// TIA Portal V20 export
TYPE "typeStationDataReelCutInspection"
   STRUCT
      "Intro cut count 1" : DInt;   // Cnt
      "Introcut Vision - Tab length 1" : Real;   // mm
      "Introcut Vision - Tab height 1" : Real;   // mm
      "Introcut Vision - Electrode length 1" : Real;   // mm
      "Introcut Vision - Electrode height 1" : Real;   // mm
      "Introcut Vision - Gap between left edge & Tab 1" : Real;   // mm
      "Introcut Vision - Gap between tab & right edge 1" : Real;   // mm
      "Introcut Vision - Height of Ceramic Coating" : Real;   // mm
      "Introcut Vision - Radii 1" : Real;   // mm
      "Introcut Vision - Height (y) of total electrode (ini. Tab) 1" : Real;   // mm
      "OK/NG" : String;   // N/A
      "Cycle end Trigger" : Bool;   // I/O
      Blocked : Bool;   // I/O
      Starved : Bool;   // I/O
      "Good Count" : DInt;   // Cnt
      "Reject Count" : DInt;   // Cnt
      "Fault bit" : Bool;   // I/O
      Fault : Bool;   // I/O
      PUN : String;   // N/A
      "FTQ & Reject code" : String;   // N/A
      "Target Cycle Time" : String;   // N/A
      "Material Low" : DInt;   // Cnt
      "2d Matrix" : String;   // N/A
      "Tool Change" : DInt;   // Cnt
   END_STRUCT;
END_TYPE
